(* IEC 61131-3 sources: com.logicals.lc3.webinar/usRTS_RPMControl_iSOC/src_FB_LIB_SAFE/Safe/Convert, 4 files *)

(* ---- wBOOL_TO_SAFEBOOL.iecst ---- *)
NAMESPACE logicals.web.standard.safe
NAMESPACE convert

/*
 * Function block wrapper for TO_SAFEBOOL<br>
 * IN =  input value (BOOL)<br>
 * OUT = IN (SAFEBOOL)<br>
 */
FUNCTION_BLOCK wBOOL_TO_SAFEBOOL
	{ vNameAlignment:="center"; altName:="BOOL_TO_SAFEBOOL"; bgColor:="Gold"; width:=160; hideIONames; }
	VAR_INPUT
		IN : BOOL;
	END_VAR
	VAR_OUTPUT
		OUT: SAFEBOOL;
	END_VAR

	IF (IN <> FALSE)
	THEN
		OUT := SAFEBOOL_Constant#SAFETRUE;
	ELSE
		OUT := SAFEBOOL_Constant#SAFEFALSE;
	END_IF;
END_FUNCTION_BLOCK

END_NAMESPACE
END_NAMESPACE

(* ---- wINT_TO_SAFEINT.iecst ---- *)
NAMESPACE logicals.web.standard.safe
NAMESPACE convert

/*
 * Function block wrapper for TO_SAFEINT<br>
 * IN =  input value (INT)<br>
 * OUT = IN (SAFEINT)<br>
 */
FUNCTION_BLOCK wINT_TO_SAFEINT
	{ vNameAlignment:="center"; altName:="INT_TO_SAFEINT"; bgColor:="GoldenRod"; width:=140; hideIONames; }
	VAR_INPUT
		IN : INT;
	END_VAR
	VAR_OUTPUT
		OUT: SAFEINT;
	END_VAR

	OUT := IN;
END_FUNCTION_BLOCK

END_NAMESPACE
END_NAMESPACE

(* ---- wSAFEBOOL_TO_BOOL.iecst ---- *)
NAMESPACE logicals.web.standard.safe
NAMESPACE convert

/*
 * Function block wrapper for TO_BOOL<br>
 * IN =  input value (SAFEBOOL)<br>
 * OUT = IN (BOOL)<br>
 */
FUNCTION_BLOCK wSAFEBOOL_TO_BOOL
	{ vNameAlignment:="center"; altName:="SAFEBOOL_TO_BOOL"; bgColor:="MediumBlue"; width:=160; hideIONames; }
	VAR_INPUT
		IN : SAFEBOOL;
	END_VAR
	VAR_OUTPUT
		OUT: BOOL;
	END_VAR

	IF (IN <> SAFEBOOL_Constant#SAFEFALSE)
	THEN
		OUT := TRUE;
	ELSE
		OUT := FALSE;
	END_IF;
	ENO := ENO AND CheckSAFEBOOL(IN);
END_FUNCTION_BLOCK

END_NAMESPACE
END_NAMESPACE

(* ---- wSAFEINT_TO_INT.iecst ---- *)
NAMESPACE logicals.web.standard.safe
NAMESPACE convert

/*
 * Function block wrapper for TO_INT<br>
 * IN =  input value (SAFEINT)<br>
 * OUT = IN (INT)<br>
 */
FUNCTION_BLOCK wSAFEINT_TO_INT
	{ vNameAlignment:="center"; altName:="SAFEINT_TO_INT"; bgColor:="LightPink"; width:=140; hideIONames; }
	VAR_INPUT
		IN : SAFEINT;
	END_VAR
	VAR_OUTPUT
		OUT: INT;
	END_VAR

	OUT := IN;
END_FUNCTION_BLOCK

END_NAMESPACE
END_NAMESPACE
